// TwinCAT 3 PLC project PLC1
// ProgramVersion: 3.1.4024.0
// libraries:
//   Tc2_ModbusRTU, * (Beckhoff Automation GmbH)
//   Tc2_Standard, * (Beckhoff Automation GmbH)
//   Tc2_System, * (Beckhoff Automation GmbH)
//   Tc3_Module, * (Beckhoff Automation GmbH)
// project tree:
//   DUTs/ E_Modbus_State.TcDUT, ST_Ecat_State.TcDUT, U_2Words_toDWord.TcDUT (not stored)
//   / PlcTask.TcTTO
//   POUs/ FB_Ecat_State.TcPOU (not stored), FB_Modbus_Rs485.TcPOU, FB_WeatherStation.TcPOU, MAIN.TcPOU
// real-time tasks:
//   TASK PlcTask: cycle T#10ms, priority 20, ADS port 350
// I/O:
//   DEVICE Device 2 (EtherCAT), AmsNetId 192.168.10.20.3.1
//     Term 1 (EK1100) [EK1100 EtherCAT Coupler (2A E-Bus)]
//       Term 2 (EL6021) [EL6021 Interface (RS422/485)]
//       Term 3 (EL6022) [EL6022 Interface 2Ch. (RS422/485)]
//       Term 4 (EL9011) [EL9011 End Terminal]
// variable links:
//   PLC1/PLC1 Instance <-> Device 2 (EtherCAT)/Term 1 (EK1100)/Term 3 (EL6022)
//     PlcTask Inputs/MAIN.fbWeatherStation.fbModbus.fbModbusMaster.InData/D <-> COM Inputs Channel 1/Data In 0
//     PlcTask Inputs/MAIN.fbWeatherStation.fbModbus.fbModbusMaster.InData/D @bit {8..168 step 8} <-> COM Inputs Channel 1/Data In {1..21}  (21 links)
//     PlcTask Inputs/MAIN.fbWeatherStation.fbModbus.fbModbusMaster.InData/Status <-> COM Inputs Channel 1/Status
//     PlcTask Inputs/MAIN.fbWeatherStation.fbModbus.fbModuleEcatState.raw_state/op_state <-> InfoData/State
//     PlcTask Inputs/MAIN.fbWeatherStation.fbModbus.fbModuleEcatState.raw_state/wc_state <-> WcState/WcState
//     PlcTask Outputs/MAIN.fbWeatherStation.fbModbus.fbModbusMaster.OutData/Ctrl <-> COM Outputs Channel 1/Ctrl
//     PlcTask Outputs/MAIN.fbWeatherStation.fbModbus.fbModbusMaster.OutData/D <-> COM Outputs Channel 1/Data Out 0
//     PlcTask Outputs/MAIN.fbWeatherStation.fbModbus.fbModbusMaster.OutData/D @bit {8..168 step 8} <-> COM Outputs Channel 1/Data Out {1..21}  (21 links)

CONFIGURATION PLC1
    RESOURCE PLC ON TwinCAT3
        TASK PlcTask(INTERVAL := T#10ms, PRIORITY := 20);
        PROGRAM MAIN WITH PlcTask : MAIN;
    END_RESOURCE
END_CONFIGURATION

// ---- DUTs/E_Modbus_State.TcDUT
// Phase 0 - E_WS_State
// Rev 1.0 - January 8, 2024

TYPE E_Modbus_State :
(
	Idle			 													:= 0,
	eReadCoils,
	ReadInputStatus,
	ReadRegs,
	ReadInputRegs,
	WriteSingleCoil,
	WriteSingleReg,
	WriteMultipleCoils,
	WriteRegs,
	Error,
	Error_Reset,
	Error_Check
);
END_TYPE

// ---- DUTs/ST_Ecat_State.TcDUT
TYPE ST_Ecat_State :
STRUCT
	wc_state : BOOL;
	op_state : UINT;
END_STRUCT
END_TYPE

// ---- POUs/MAIN.TcPOU
PROGRAM MAIN
VAR
	fbWeatherStation : FB_WeatherStation;
END_VAR

fbWeatherStation();

END_PROGRAM

// ---- POUs/FB_WeatherStation.TcPOU
FUNCTION_BLOCK FB_WeatherStation
VAR_INPUT
END_VAR
VAR_OUTPUT
	o_press_Pa : REAL ;
	o_temp_degc : REAL;
	o_humidity_rh : REAL;
	o_wind_direction_deg : REAL;
	o_wind_speed_ms : REAL;
	o_dew_point_degC : REAL;
END_VAR
VAR
	fbModbus : FB_Modbus_Rs485;
	raw_data : ARRAY[0..25] OF WORD;
	modbus_error : BOOL;
	
	raw_pressure :  U_2Words_toDWord;
	
END_VAR

fbModbus(
	i_slave_id:= 1, 
	i_start_read_address:= 1,
	i_registers_qty := 23, 
	o_error=> modbus_error, 
	io_raw_data:= raw_data);

o_temp_degc := TO_REAL(raw_data[0])/10;
o_humidity_rh := TO_REAL(raw_data[1])/10;
o_wind_direction_deg := TO_REAL(raw_data[2]);
o_wind_speed_ms := TO_REAL(raw_data[3])/10;
o_dew_point_degC := TO_REAL(raw_data[18])/10;


	
	
raw_pressure.u_words[1] := raw_data[11];
raw_pressure.u_words[0] := raw_data[12];
o_press_Pa := TO_REAL(raw_pressure.u_dword)/10;

END_FUNCTION_BLOCK

// ---- POUs/FB_Modbus_Rs485.TcPOU
FUNCTION_BLOCK FB_Modbus_Rs485
VAR_INPUT
	i_slave_id		 	 	: BYTE;
	i_start_read_address 	: WORD;
	i_registers_qty			: WORD;
		  
END_VAR
	
VAR_OUTPUT
	o_error : BOOL;
END_VAR

VAR_IN_OUT
	io_raw_data		: ARRAY[*] OF WORD;	
END_VAR

VAR
	fbModuleEcatState : FB_Ecat_State;
	
	fbModbusMaster 														: ModbusRtuMasterV2_KL6x22B;	
	modbus_state														: E_Modbus_State;
	raw_data_read 														: ARRAY[0..100] OF WORD;
	_TIMEOUT_MODBUS														: TIME 		:= T#2S;
	
	size_local_array :  UINT;
	size_io_array : UINT;
	idxReg : DINT;
	error_modbus : BOOL;
	error_id : MODBUS_ERRORS;
END_VAR


CASE modbus_state OF
	
	E_Modbus_State.Idle:
		fbModbusMaster.Execute := FALSE;
		
		IF NOT o_error THEN
			modbus_state := E_Modbus_State.ReadRegs;
		END_IF
		
	E_Modbus_State.ReadRegs:
		fbModbusMaster.ReadRegs(Execute := TRUE);
		IF NOT fbModbusMaster.BUSY  AND NOT fbModbusMaster.Error THEN
					fbModbusMaster.ReadRegs(Execute := FALSE);
		ELSIF fbModbusMaster.Error THEN	  
					modbus_state := E_Modbus_State.Error;				
		END_IF	
		
	E_Modbus_State.Error :
		 error_modbus := TRUE;
		 fbModbusMaster.Execute := FALSE;	
		 modbus_state := E_Modbus_State.Error_Reset;
		 
	E_Modbus_State.Error_Reset :
		fbModbusMaster.Execute := TRUE;
		IF NOT fbModbusMaster.BUSY AND NOT fbModbusMaster.Error THEN
			error_modbus := FALSE;
			modbus_state := E_Modbus_State.Idle;
		ELSE
			modbus_state := E_Modbus_State.Error;
		END_IF
		
			
	
END_CASE

fbModbusMaster.ReadRegs(UnitID 			:= i_slave_id,
					   Quantity			:= i_registers_qty, 
					   MBAddr			:= i_start_read_address, 
					   cbLength			:= SIZEOF(raw_data_read), 
					   pMemoryAddr		:= ADR(raw_data_read), 
					   Timeout			:= _TIMEOUT_MODBUS);


FOR idxReg := LOWER_BOUND(io_raw_data,1) TO UPPER_BOUND(io_raw_data,1) DO 
	io_raw_data[idxReg] := raw_data_read[idxReg];
END_FOR


o_error  := NOT fbModuleEcatState.State OR error_modbus ;

END_FUNCTION_BLOCK
